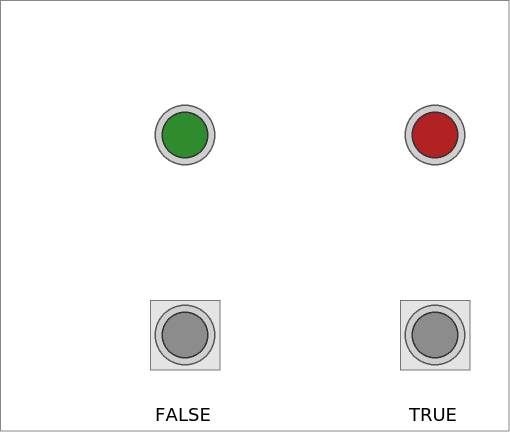
VISUALIZATION Visualization  // 510x432
    PushSwitch (150,300 70x70), tooltip "FALSE", variable: GVL_IO.b_blue_button, behaviour: TOGGLE, style: Switch-PushSwitch-Gray
    PushSwitch (400,300 70x70), tooltip "TRUE", variable: GVL_IO.b_yellow_button, behaviour: TOGGLE, style: Switch-PushSwitch-Gray
    Lamp1 (150,100 70x70), variable: GVL_IO.b_green_lamp, style: Lamp-Lamp1-Green
    Lamp1 (400,100 70x70), variable: GVL_IO.b_red_lamp, style: Lamp-Lamp1-Red
    Label (108,400 150x30), "FALSE"
    Label (358,400 150x30), "TRUE"
END_VISUALIZATION

(* stored: Version 1.1.0.1, ProductVersion 3.1.4022.12
   Visu Visualization: Id {5dc87ccc-885e-4dda-a8cc-555f27963805} *)
